(* PLC project SansNom, Inconnu SansNom 1 *)
(* stored: creationDateTime 2026-08-12T11:47:00, modificationDateTime 2026-08-13T12:11:19 *)

PROGRAM program0
  VAR
    AUTO AT %IX0.0 : BOOL;  (* Interrupteur maintenu du mode automatique en boucle *)
    BPON AT %IX0.1 : BOOL;  (* Poussoir : lance un cycle unique *)
    BPOFF AT %IX0.2 : BOOL;  (* Poussoir : demande l'arrêt du mode auto (effectif en fin de cycle) *)
    LED1 AT %QX0.0 : BOOL;  (* Voyant 1 *)
    LED2 AT %QX0.1 : BOOL;  (* Voyant 2 *)
    LED3 AT %QX0.2 : BOOL;  (* Voyant 3 *)
    LED4 AT %QX0.3 : BOOL;  (* Voyant 4 *)
    Demande_arret AT %MX0.3 : BOOL := FALSE;  (* Mémorise l'appui sur BPOFF jusqu'à la fin du cycle en cours *)
    Inhibition_auto AT %MX0.4 : BOOL := FALSE;  (* Empêche un redémarrage auto immédiat après un arrêt BPOFF tant que AUTO reste à 1 *)
    Va1 AT %MX0.0 : BOOL := FALSE;  (* Variable auxiliaire 1 *)
    Va2 AT %MX0.1 : BOOL := FALSE;  (* Variable auxiliaire 2 *)
    tout_eteint AT %MX0.2 : BOOL := FALSE;  (* Variable auxiliaire 2 *)
    T8_done AT %MX0.3 : BOOL;  (* Reçoit la sortie Q de T8 *)
  END_VAR
  VAR
    Tempo : TIME := T#500ms;
    TON0 : TON;
    TON1 : TON;
    TON2 : TON;
    TON3 : TON;
    TON4 : TON;
    TON5 : TON;
    TON6 : TON;
    TON7 : TON;
    TON8 : TON;
  END_VAR
  VAR  (* added by the conversion: wires and edge detectors of the diagram *)
    F_TRIG1 : F_TRIG;
    F_TRIG2 : F_TRIG;
  END_VAR

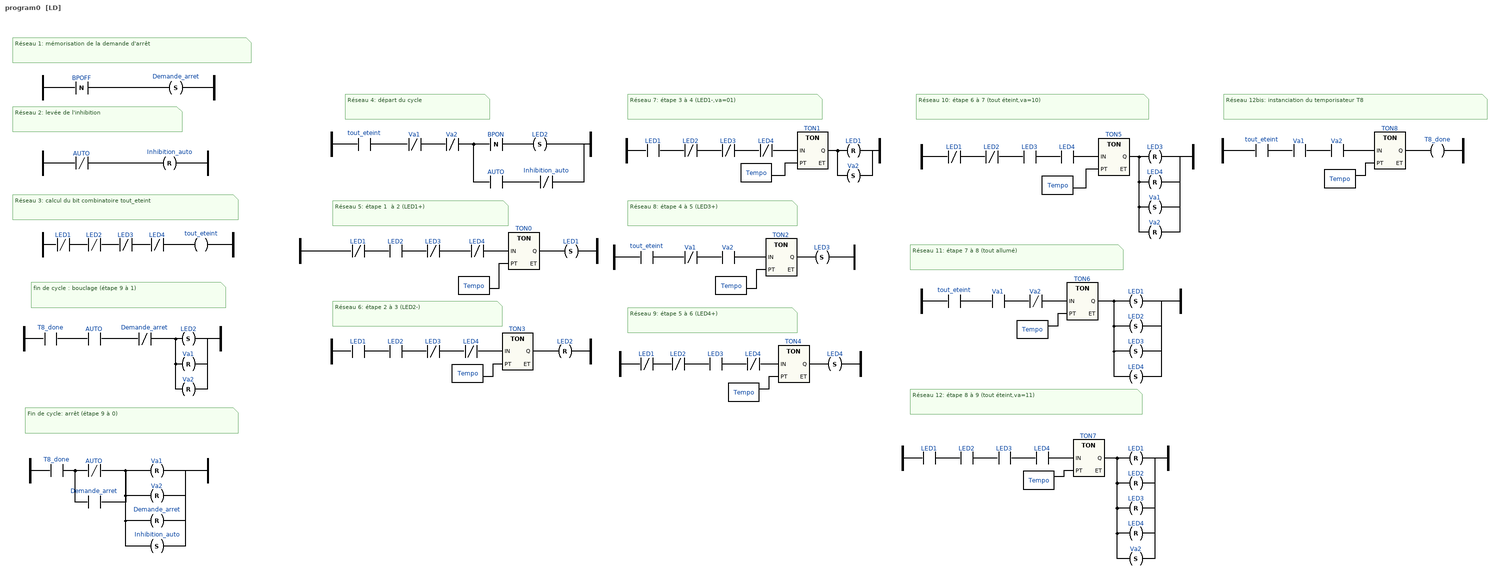
(* LD diagram, written out as Structured Text *)
(* Réseau 1: mémorisation de la demande d'arrêt *)
F_TRIG1(CLK := BPOFF);
IF F_TRIG1.Q THEN Demande_arret := TRUE; END_IF;
(* Réseau 4: départ du cycle *)
(* Réseau 7: étape 3 à 4 (LED1-,va=01) *)
(* Réseau 10: étape 6 à 7 (tout éteint,va=10) *)
(* Réseau 12bis: instanciation du temporisateur T8 *)
(* Réseau 2: levée de l'inhibition *)
IF NOT AUTO THEN Inhibition_auto := FALSE; END_IF;
(* Réseau 3: calcul du bit combinatoire tout_eteint *)
(* Réseau 5: étape 1  à 2 (LED1+) *)
(* Réseau 8: étape 4 à 5 (LED3+) *)
tout_eteint := NOT LED1 AND NOT LED2 AND NOT LED3 AND NOT LED4;
F_TRIG2(CLK := BPON);
IF tout_eteint AND NOT Va1 AND NOT Va2 AND F_TRIG2.Q THEN LED2 := TRUE; END_IF;
(* Réseau 11: étape 7 à 8 (tout allumé) *)
TON0(IN := NOT LED1 AND LED2 AND NOT LED3 AND NOT LED4, PT := Tempo);
IF TON0.Q THEN LED1 := TRUE; END_IF;
(* fin de cycle : bouclage (étape 9 à 1) *)
(* Réseau 6: étape 2 à 3 (LED2-) *)
(* Réseau 9: étape 5 à 6 (LED4+) *)
TON3(IN := LED1 AND LED2 AND NOT LED3 AND NOT LED4, PT := Tempo);
IF TON3.Q THEN LED2 := FALSE; END_IF;
TON1(IN := LED1 AND NOT LED2 AND NOT LED3 AND NOT LED4, PT := Tempo);
IF TON1.Q THEN LED1 := FALSE; END_IF;
IF TON1.Q THEN Va2 := TRUE; END_IF;
TON2(IN := tout_eteint AND NOT Va1 AND Va2, PT := Tempo);
IF TON2.Q THEN LED3 := TRUE; END_IF;
TON4(IN := NOT LED1 AND NOT LED2 AND LED3 AND NOT LED4, PT := Tempo);
IF TON4.Q THEN LED4 := TRUE; END_IF;
TON5(IN := NOT LED1 AND NOT LED2 AND LED3 AND LED4, PT := Tempo);
IF TON5.Q THEN LED3 := FALSE; END_IF;
IF TON5.Q THEN LED4 := FALSE; END_IF;
IF TON5.Q THEN Va1 := TRUE; END_IF;
IF TON5.Q THEN Va2 := FALSE; END_IF;
TON6(IN := tout_eteint AND Va1 AND NOT Va2, PT := Tempo);
IF TON6.Q THEN LED1 := TRUE; END_IF;
IF TON6.Q THEN LED2 := TRUE; END_IF;
IF TON6.Q THEN LED3 := TRUE; END_IF;
IF TON6.Q THEN LED4 := TRUE; END_IF;
(* Réseau 12: étape 8 à 9 (tout éteint,va=11) *)
(* Fin de cycle: arrêt (étape 9 à 0) *)
TON7(IN := LED1 AND LED2 AND LED3 AND LED4, PT := Tempo);
IF TON7.Q THEN LED1 := FALSE; END_IF;
IF TON7.Q THEN LED2 := FALSE; END_IF;
IF TON7.Q THEN LED3 := FALSE; END_IF;
IF TON7.Q THEN LED4 := FALSE; END_IF;
IF TON7.Q THEN Va2 := TRUE; END_IF;
IF T8_done AND AUTO AND NOT Demande_arret THEN LED2 := TRUE; END_IF;
IF T8_done AND AUTO AND NOT Demande_arret THEN Va1 := FALSE; END_IF;
IF T8_done AND AUTO AND NOT Demande_arret THEN Va2 := FALSE; END_IF;
TON8(IN := tout_eteint AND Va1 AND Va2, PT := Tempo);
T8_done := TON8.Q;
IF T8_done AND (NOT AUTO OR Demande_arret) THEN Va1 := FALSE; END_IF;
IF T8_done AND NOT AUTO THEN Va2 := FALSE; END_IF;
IF T8_done AND NOT AUTO THEN Demande_arret := FALSE; END_IF;
IF T8_done AND NOT AUTO THEN Inhibition_auto := TRUE; END_IF;
(* drawn but not wired to any output: AUTO, Inhibition_auto *)
END_PROGRAM

CONFIGURATION Config0
  RESOURCE Res0 ON PLC
    TASK task0(INTERVAL := T#20ms, PRIORITY := 0);
    PROGRAM instance0 WITH task0 : program0;
  END_RESOURCE
END_CONFIGURATION
